FUNCTION_BLOCK FB_Unit IMPLEMENTS ITF_UnitState
VAR_INPUT (*  	Remark: Since the structure is not implemented as nested FB instances
				the status tags cannot be protected against external manipulation (read-only)
				thus they shall be overwritten each cycle to keep consistancy 			
		
				Could also be mitigated if proper OPC UA pragmas were applied
				within the structure - would require redefinition of top-level
				struct below 
				*)
	{attribute 'TcAnalytics'}
	{attribute 'OPC.UA.DA' := '1'}	
	stPackTags	: ST_PML_Custom;		// Custom pack tags from project
END_VAR

VAR (* 	Protected internal status
		not accessibly, invisible 
		*)
	{attribute 'hide'}
	nMode	: DINT := E_PMLMode.UNDEFINED; // Actual mode of the Unit
	
	{attribute 'hide'}
	bModeValid : BOOL := FALSE; // Indicate if a valid mode is set
	
	{attribute 'hide'}
	eState	: E_PMLState := ePMLState_Aborted; // Actual state of the Unit
	
	{attribute 'hide'}
	fSpeed_Set : REAL; // Set-value of the machine speed
	
	{attribute 'hide'}
	fSpeed_Act : REAL; // Act-value of the machine speed
END_VAR

VAR (*	Mode handler variables *)
	
	{attribute 'hide'}
	fbModeManager : PML_UnitModeManager; // Encapsulated mode change logic
	
	{attribute 'hide'}
	eModeHandler_State : (Wait_For_Change_Request, Switch_Mode, Report_Error); // Method state machine
END_VAR

VAR (*	State handler variables *)
	
	{attribute 'hide'}
	fbStateManager : PML_StateMachine;
END_VAR

(* Refesh the status tags *)
SetTags();

(* Handle mode requests and perform changes *)
ModeHandler();

(* Handle the state if in an valid mode *)
IF bModeValid THEN
	StateHandler();
END_IF

(* Handle the speed request *)
SpeedHandler();

{attribute 'object_name' := 'M_Aborted'}
METHOD M_Aborted
END_METHOD

{attribute 'object_name' := 'M_Aborting'}
METHOD M_Aborting
stPackTags.Admin.StopReason[1].ID := E_PMLStopReason.Abort_User;
M_StateComplete();
END_METHOD

{attribute 'object_name' := 'M_Clearing'}
METHOD M_Clearing
M_StateComplete();
END_METHOD

{attribute 'object_name' := 'M_Complete'}
METHOD M_Complete
END_METHOD

{attribute 'object_name' := 'M_Completing'}
METHOD M_Completing
M_StateComplete();
END_METHOD

{attribute 'object_name' := 'M_Execute'}
METHOD M_Execute
END_METHOD

{attribute 'object_name' := 'M_Held'}
METHOD M_Held
END_METHOD

{attribute 'object_name' := 'M_Holding'}
METHOD M_Holding
stPackTags.Admin.StopReason[1].ID:= E_PMLStopReason.Held_Ingredients;
M_StateComplete();
END_METHOD

{attribute 'object_name' := 'M_Idle'}
METHOD M_Idle
END_METHOD

{attribute 'object_name' := 'M_Resetting'}
METHOD M_Resetting
stPackTags.Admin.StopReason[1].ID:= E_PMLStopReason.None;
stPackTags.Status.EquipmentInterlock.Blocked := FALSE;
stPackTags.Status.EquipmentInterlock.Starved := FALSE;
M_StateComplete();
END_METHOD

{attribute 'object_name' := 'M_Starting'}
METHOD M_Starting
M_StateComplete();
END_METHOD

{attribute 'object_name' := 'M_StateComplete'}
METHOD M_StateComplete
//the actual state is completed
fbStateManager.M_StateComplete();
END_METHOD

{attribute 'object_name' := 'M_Stopped'}
METHOD M_Stopped
END_METHOD

{attribute 'object_name' := 'M_Stopping'}
METHOD M_Stopping
stPackTags.Admin.StopReason[1].ID := E_PMLStopReason.Stop_Actuators;
M_StateComplete();
END_METHOD

{attribute 'object_name' := 'M_Suspended'}
METHOD M_Suspended
END_METHOD

{attribute 'object_name' := 'M_Suspending'}
METHOD M_Suspending
stPackTags.Admin.StopReason[1].ID := E_PMLStopReason.Suspend_Blocked;
stPackTags.Status.EquipmentInterlock.Blocked := TRUE;
M_StateComplete();
END_METHOD

{attribute 'object_name' := 'M_Undefined'}
METHOD M_Undefined
END_METHOD

{attribute 'object_name' := 'M_Unholding'}
METHOD M_Unholding
stPackTags.Admin.StopReason[1].ID := E_PMLStopReason.None;
M_StateComplete();
END_METHOD

{attribute 'object_name' := 'M_Unsuspending'}
METHOD M_Unsuspending
stPackTags.Admin.StopReason[1].ID := E_PMLStopReason.None;
stPackTags.Status.EquipmentInterlock.Blocked := FALSE;
M_StateComplete();
END_METHOD

{attribute 'object_name' := 'ModeHandler'}
METHOD PROTECTED ModeHandler
CASE eModeHandler_State OF
	Wait_For_Change_Request:
		IF stPackTags.Command.UnitModeChangeRequest = TRUE
		AND stPackTags.Command.UnitMode <> E_PMLMode.UNDEFINED
		AND stPackTags.Command.UnitMode <> nMode THEN
			bModeValid := FALSE;
			fbModeManager.eModeCommand := stPackTags.Command.UnitMode;
			eModeHandler_State := Switch_Mode;
		END_IF
		
	Switch_Mode:
		fbModeManager.bExecute := TRUE;
		
		IF fbModeManager.bDone THEN
			bModeValid := TRUE;
			fbModeManager.bExecute := FALSE;
			eModeHandler_State := Wait_For_Change_Request;
			
		ELSIF fbModeManager.bError THEN
			fbModeManager.bExecute := FALSE;
			eModeHandler_State := Report_Error;
		END_IF
		
	Report_Error:
		;
		// Set the machine on fire to highlight urgency
END_CASE

(* 	Execute the mode manager
	and update the status*)
fbModeManager( eState := eState, eModeStatus => nMode);
stPackTags.Status.UnitModeCurrent := nMode;
END_METHOD

{attribute 'object_name' := 'SetTags'}
METHOD PROTECTED SetTags
VAR_INPUT
END_VAR
stPackTags.Status.MachineSpeed := 100;
stPackTags.Status.CurMachineSpeed := 0;
stPackTags.Status.UnitModeCurrent := 0;
END_METHOD

{attribute 'object_name' := 'SpeedHandler'}
METHOD PROTECTED SpeedHandler
VAR_INPUT
END_VAR
(* 	Leave if machine speed mateches the request *)
IF fSpeed_Set = stPackTags.Command.MachSpeed THEN
	RETURN;
END_IF

(*	Apply machine speed within the machines limitations *)
IF stPackTags.Command.MachSpeed <= stPackTags.Status.MachineSpeed THEN
	fSpeed_Set := stPackTags.Command.MachSpeed;
ELSE
	fSpeed_Set := stPackTags.Status.MachineSpeed;
END_IF
END_METHOD

{attribute 'object_name' := 'StateHandler'}
METHOD PROTECTED StateHandler
IF stPackTags.Command.CmdChangeRequest = TRUE THEN
	(* 	Execute the state manager
		and update the status *)
	fbStateManager(eMode	:= nMode, eCommand := stPackTags.Command.CntrlCmd, eState	=> eState);
	stPackTags.Status.StateCurrent := eState;
END_IF

IF stPackTags.Status.UnitModeCurrent <> E_PMLMode.UNDEFINED AND stPackTags.Status.StateCurrent = E_PMLState.ePMLState_Undefined THEN
	stPackTags.Command.CmdChangeRequest := TRUE;
	fbStateManager(eMode	:= nMode, eCommand := E_PMLCommand.ePMLCommand_Abort, eState => eState);
END_IF

IF fbStateManager.bError THEN
	// Set the machine on fire to highlight urgency
END_IF

(*	Process the state method *)
CASE eState OF
	ePMLState_Undefined: M_Undefined();
	ePMLState_Clearing: M_Clearing();
	ePMLState_Stopped: M_Stopped();
	ePMLState_Starting: M_Starting();
	ePMLState_Idle: M_Idle();
	ePMLState_Suspended: M_Suspended();
	ePMLState_Execute: M_Execute();
	ePMLState_Stopping: M_Stopping();
	ePMLState_Aborting: M_Aborting();
	ePMLState_Aborted: M_Aborted();
	ePMLState_Holding: M_Holding();
	ePMLState_Held: M_Held();
	ePMLState_Unholding: M_Unholding();
	ePMLState_Suspending: M_Suspending();
	ePMLState_Unsuspending: M_Unsuspending();
	ePMLState_Resetting: M_Resetting();
	ePMLState_Completing: M_Completing();
	ePMLState_Complete: M_Complete();
END_CASE
END_METHOD

END_FUNCTION_BLOCK

(* stored: Version 1.1.0.1, ProductVersion 3.1.4024.13
   POU FB_Unit: Id {410e3470-878d-4722-b65d-1220314c3a74}, SpecialFunc None
   Folder Handler: Id {8bdb4209-4292-4a31-a723-2ef5e204b684}
   Folder States: Id {7ff35325-bdb9-41bd-ab67-f01c141199d6}
   Method M_Aborted: Id {b038fdd7-dc6d-44a1-b397-7029d2ebf77c}
   Method M_Aborting: Id {730cefcd-cd98-4ab4-8cb2-9b51dd737779}
   Method M_Clearing: Id {e2f89338-466a-4bce-bc2d-28329c1ea40c}
   Method M_Complete: Id {c7286240-808e-43c2-b4a0-1cb71c917780}
   Method M_Completing: Id {3865d34a-95bb-489e-a80f-f56cef99e355}
   Method M_Execute: Id {4a4a6499-77d3-41d8-83ad-21f487ab1083}
   Method M_Held: Id {35127f11-b6c7-4319-beb1-413d37338461}
   Method M_Holding: Id {c1185b9a-80dd-4e1d-8924-1bcd7dbed3e7}
   Method M_Idle: Id {e9ef96f0-6e56-40ed-89c6-f74cc6b7d852}
   Method M_Resetting: Id {7402e195-41c6-42ba-ab78-3c23871ffe13}
   Method M_Starting: Id {a18f3c3b-96d1-4ec2-aa4e-5dca8bef7706}
   Method M_StateComplete: Id {7d74670e-e4f1-4d4a-b620-229506688540}
   Method M_Stopped: Id {7f19ec1b-4b69-4891-b5c4-158723ccb71d}
   Method M_Stopping: Id {9cb5cdb2-58c0-4739-9252-5d901726de03}
   Method M_Suspended: Id {ad3de43a-4758-4379-bb77-abed2ae62a38}
   Method M_Suspending: Id {ed176e6f-51a2-4ef8-8404-62a78e9e476c}
   Method M_Undefined: Id {70548b7d-d2ff-4b24-9935-909058aded4e}
   Method M_Unholding: Id {5b5c8001-7d7e-433e-bcbe-af8e8200d71b}
   Method M_Unsuspending: Id {bba01a33-53b5-47e4-a67f-889524fcf7b8}
   Method ModeHandler: Id {ac7899a8-1526-4955-a4d2-c36a7f77b10b}
   Method SetTags: Id {3b37a057-96f9-4024-8c89-2f6438a0cedd}
   Method SpeedHandler: Id {cd4a2691-959e-4109-8922-b0efd7e25427}
   Method StateHandler: Id {2a53a776-d2a2-499e-8b47-a2228820e21e} *)
